PROGRAM PRG_TimestampRegistry
VAR 
	fbReadTime				:FB_ReadTime;	
	bSignalIn				:BOOL;
	bReset					:BOOL;
END_VAR

//Set Commands
M_SetCommands();


//Call read time
fbReadTime(bReset := bReset,
		   bSignalIn := bSignalIn);


//Reset Commands
M_ResetCommands();

METHOD PRIVATE M_ResetCommands
VAR_INPUT
END_VAR
//Reset Commands
GVL_HMI.stTimestampCmd.bResetRegistry := FALSE;
END_METHOD

METHOD PRIVATE M_SetCommands
VAR_INPUT
END_VAR
//Set Commands
bReset := GVL_HMI.stTimestampCmd.bResetRegistry;
bSignalIn := GVL_IO.stItemSimulator.bSignalIn;
END_METHOD

METHOD PUBLIC M_StatusHMI
VAR_INPUT
END_VAR
END_METHOD

END_PROGRAM

(* stored: Version 1.1.0.1, ProductVersion 3.1.4024.12
   POU PRG_TimestampRegistry: Id {41809a93-5b53-47f0-b8b5-05c700b2cea3}, SpecialFunc None
   Method M_ResetCommands: Id {74db0409-a38e-4eee-b70a-2501178068c0}
   Method M_SetCommands: Id {51730a3a-dc77-4efb-ad56-60c19693c631}
   Method M_StatusHMI: Id {07c83b8d-d512-478b-acd0-c9301802f0e4} *)
